(* CoDeSys 2.3.9.37 project: Cap6_8.pro *)
(* Libraries: Standard.lib 4.10.05 12:14:46 *)

(* Global variable list: Global_Variables *)
VAR_GLOBAL

 (* Entradas *)
  A:BOOL;
  B:BOOL;
  C:BOOL;

(* Salidas *)
  SAL:BOOL;

END_VAR

(* POU PLC_PRG, LD *)
PROGRAM PLC_PRG
VAR
END_VAR
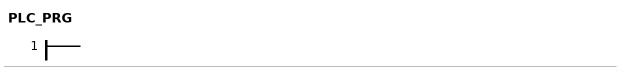
_LD_ (* Ladder Diagram *)
NETWORK 1
	*
_END_LD_
(* the same logic as Structured Text *)
(* Network 1 *)
END_PROGRAM

(* Visualisation Visio
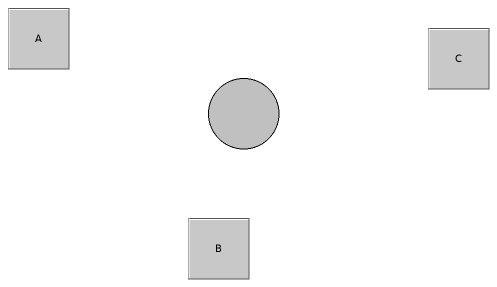
button at (80,40)-(141,101): text "A"; toggles A
button at (500,60)-(561,121): text "C"; toggles C
button at (260,250)-(321,311): text "B"; toggles B
ellipse at (280,110)-(351,181): alarm colour if SAL
*)
